Yaskawa INFORM job: BUFFER_INIT.JBI

/JOB
//NAME BUFFER_INIT
//POS
///NPOS 0,0,0,0,0,0
//INST
///DATE 2011/12/02 15:43
///ATTR SC,RW
///GROUP1 RB1
NOP
SET I091 0
SET I092 0
WHILE I092<=I093
	 WAIT B000<>0 T=0.10
ENDWHILE
END
